TYPE HMI_SP_TemplateClean :
STRUCT
	CFG_MachinePartEnabled:BOOL:=TRUE;				(*Configuration this machinepart is enabled >> when disabled I_SN_SUP_Request is coupled directly to Q_SN_DSC_Request and errors+organiser stuff is put in the correct state*)
	
END_STRUCT
END_TYPE

(* stored: Version 1.1.0.1, ProductVersion 3.1.4024.3
   DUT HMI_SP_TemplateClean: Id {fa7b424d-320a-46fe-aa94-64457783369a} *)
